// TwinCAT 3 PLC project Style1
// ProgramVersion: 1.0.0.0
// libraries:
//   Tc2_Standard, * (Beckhoff Automation GmbH)
//   Tc2_System, * (Beckhoff Automation GmbH)
//   Tc3_GlobalTypes
//   Tc3_Module, * (Beckhoff Automation GmbH)
// project tree:
//   / PlcTask.TcTTO
//   POUs/ A_Program.TcPOU, B_Program.TcPOU, MAIN.TcPOU
// real-time tasks:
//   TASK PlcTask: cycle T#10ms, priority 20, ADS port 350
//   TASK PlcTask1: cycle T#10ms, priority 21, ADS port 351

CONFIGURATION Style1
    RESOURCE PLC ON TwinCAT3
        TASK PlcTask(INTERVAL := T#10ms, PRIORITY := 20);
        PROGRAM MAIN WITH PlcTask : MAIN;
    END_RESOURCE
END_CONFIGURATION

// ---- POUs/MAIN.TcPOU
PROGRAM MAIN
VAR
END_VAR

A_Program();

END_PROGRAM

// ---- POUs/A_Program.TcPOU
PROGRAM A_Program
VAR
END_VAR

B_Program();

END_PROGRAM

// ---- POUs/B_Program.TcPOU
PROGRAM B_Program
VAR
	i : UINT;
	x : LREAL;
	x_inc : LREAL := 0.0001;
END_VAR

FOR i := 0 TO 100 DO
	x := x + x_inc;
END_FOR

END_PROGRAM
